// TIA Portal V17 program export: 1 tag tables, 0 data types, 0 data blocks, 2 code blocks (in call order from the OBs), 0 instance data blocks

VAR_GLOBAL   // PLC tag table "Default tag table"
   "jaw latch" AT %M0.0 : Bool;
   "jaw output" AT %M0.1 : Bool;
   "prog reset" AT %M0.2 : Bool;
   TempVar AT %MW2 : Word;
   AlwaysOn AT %M0.3 : Bool;
   StartLatch AT %M0.4 : Bool;
   StartLatchBit AT %M0.5 : Bool;
END_VAR

ORGANIZATION_BLOCK "Main"   // OB1, LAD, ProgramCycle
TITLE = "Main Program Sweep (Cycle)"
{ S7_Optimized_Access := 'TRUE' }
VERSION : 0.1
// stored: AutoNumber true, IsIECCheckEnabled false, SetENOAutomatically false
   VAR_INPUT
      Initial_Call : Bool;   // Initial call of this OB
      Remanence : Bool;   // =True, if remanent data are available
   END_VAR
BEGIN

REGION Network 1
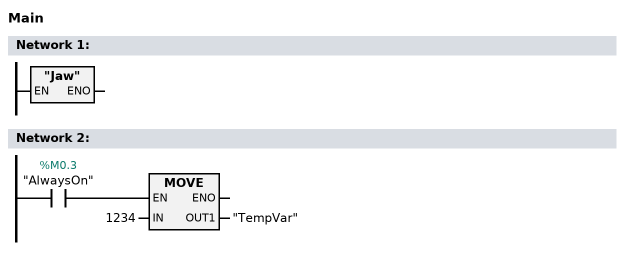
   RUNG wire#powerrail
      "Jaw"()
   END_RUNG
   // the same network as SCL:
   "Jaw"();
END_REGION

REGION Network 2
   RUNG wire#powerrail
      Contact( "AlwaysOn" )
      Move(in := 1234, out1 => "TempVar")
   END_RUNG
   // the same network as SCL:
   IF "AlwaysOn" THEN "TempVar" := 1234; END_IF;
END_REGION
END_ORGANIZATION_BLOCK

FUNCTION "Jaw" : Void   // FC1, LAD
{ S7_Optimized_Access := 'TRUE' }
VERSION : 0.1
// stored: AutoNumber true, IsIECCheckEnabled false, SetENOAutomatically false, UDAEnableTagReadback false
BEGIN

REGION Network 1
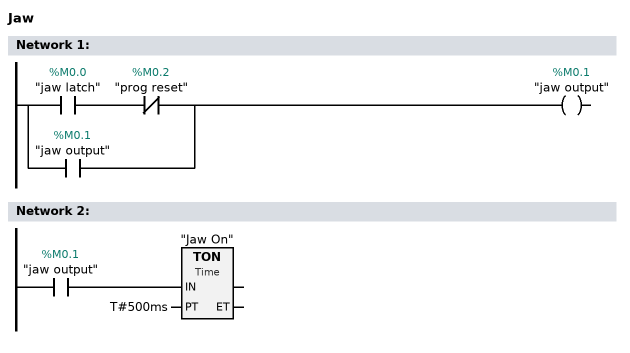
   RUNG wire#powerrail
      Contact( "jaw latch" )
      I_Contact( "prog reset" )
      wire#w1
      Coil( "jaw output" )
   END_RUNG
   RUNG wire#powerrail
      Contact( "jaw output" )
   END_RUNG wire#w1
   // the same network as SCL:
   "jaw output" := ("jaw latch" AND NOT "prog reset") OR "jaw output";
END_REGION

REGION Network 2
   RUNG wire#powerrail
      Contact( "jaw output" )
      { S7_Templates := "time_type := Time" } "Jaw On".TON(pt := T#500ms, et =>)
   END_RUNG
   // the same network as SCL:
   "Jaw On".TON(IN := "jaw output", PT := T#500ms);
END_REGION
END_FUNCTION
